{attribute addProperty BoxType "EJ6002-0000-0016"}
{attribute addProperty Id "StatusAT %I*Status_0CBEDEF81621Data_InAT %I*ARRAY[0 ..21] OF USINT176220"}
{attribute addProperty CRC "3699519399"}
{attribute addProperty SizeInBites "192"}
{attribute addProperty SizeInBytes "24"}
TYPE COM_Inputs_Channel_85D1D733 :
STRUCT
	{attribute addProperty Name "Status"}
	Status AT %I* : Status_0CBEDEF8;
	{attribute addProperty Name "Data_In"}
	Data_In AT %I* : ARRAY[0 ..21] OF USINT;
END_STRUCT
END_TYPE

(* stored: Version 1.2.0.0, ProductVersion 3.1.4024.9
   DUT COM_Inputs_Channel_85D1D733: Id {d66bb796-710a-49f5-b87c-623a7bb2dce3} *)
